  965 = 'S4_Warnings Default 965' | German: 'S4_Warnings German 965' | French: 'S4_Warnings French 965'
  966 = 'S4_Warnings Default 966' | German: 'S4_Warnings German 966' | French: 'S4_Warnings French 966'
  967 = 'S4_Warnings Default 967' | German: 'S4_Warnings German 967' | French: 'S4_Warnings French 967'
  968 = 'S4_Warnings Default 968' | German: 'S4_Warnings German 968' | French: 'S4_Warnings French 968'
  969 = 'S4_Warnings Default 969' | German: 'S4_Warnings German 969' | French: 'S4_Warnings French 969'
  970 = 'S4_Warnings Default 970' | German: 'S4_Warnings German 970' | French: 'S4_Warnings French 970'
  971 = 'S4_Warnings Default 971' | German: 'S4_Warnings German 971' | French: 'S4_Warnings French 971'
  972 = 'S4_Warnings Default 972' | German: 'S4_Warnings German 972' | French: 'S4_Warnings French 972'
  973 = 'S4_Warnings Default 973' | German: 'S4_Warnings German 973' | French: 'S4_Warnings French 973'
  974 = 'S4_Warnings Default 974' | German: 'S4_Warnings German 974' | French: 'S4_Warnings French 974'
  975 = 'S4_Warnings Default 975' | German: 'S4_Warnings German 975' | French: 'S4_Warnings French 975'
  976 = 'S4_Warnings Default 976' | German: 'S4_Warnings German 976' | French: 'S4_Warnings French 976'
  977 = 'S4_Warnings Default 977' | German: 'S4_Warnings German 977' | French: 'S4_Warnings French 977'
  978 = 'S4_Warnings Default 978' | German: 'S4_Warnings German 978' | French: 'S4_Warnings French 978'
  979 = 'S4_Warnings Default 979' | German: 'S4_Warnings German 979' | French: 'S4_Warnings French 979'
  980 = 'S4_Warnings Default 980' | German: 'S4_Warnings German 980' | French: 'S4_Warnings French 980'
  981 = 'S4_Warnings Default 981' | German: 'S4_Warnings German 981' | French: 'S4_Warnings French 981'
  982 = 'S4_Warnings Default 982' | German: 'S4_Warnings German 982' | French: 'S4_Warnings French 982'
  983 = 'S4_Warnings Default 983' | German: 'S4_Warnings German 983' | French: 'S4_Warnings French 983'
  984 = 'S4_Warnings Default 984' | German: 'S4_Warnings German 984' | French: 'S4_Warnings French 984'
  985 = 'S4_Warnings Default 985' | German: 'S4_Warnings German 985' | French: 'S4_Warnings French 985'
  986 = 'S4_Warnings Default 986' | German: 'S4_Warnings German 986' | French: 'S4_Warnings French 986'
  987 = 'S4_Warnings Default 987' | German: 'S4_Warnings German 987' | French: 'S4_Warnings French 987'
  988 = 'S4_Warnings Default 988' | German: 'S4_Warnings German 988' | French: 'S4_Warnings French 988'
  989 = 'S4_Warnings Default 989' | German: 'S4_Warnings German 989' | French: 'S4_Warnings French 989'
  990 = 'S4_Warnings Default 990' | German: 'S4_Warnings German 990' | French: 'S4_Warnings French 990'
  991 = 'S4_Warnings Default 991' | German: 'S4_Warnings German 991' | French: 'S4_Warnings French 991'
  992 = 'S4_Warnings Default 992' | German: 'S4_Warnings German 992' | French: 'S4_Warnings French 992'
  993 = 'S4_Warnings Default 993' | German: 'S4_Warnings German 993' | French: 'S4_Warnings French 993'
  994 = 'S4_Warnings Default 994' | German: 'S4_Warnings German 994' | French: 'S4_Warnings French 994'
  995 = 'S4_Warnings Default 995' | German: 'S4_Warnings German 995' | French: 'S4_Warnings French 995'
  996 = 'S4_Warnings Default 996' | German: 'S4_Warnings German 996' | French: 'S4_Warnings French 996'
  997 = 'S4_Warnings Default 997' | German: 'S4_Warnings German 997' | French: 'S4_Warnings French 997'
  998 = 'S4_Warnings Default 998' | German: 'S4_Warnings German 998' | French: 'S4_Warnings French 998'
  999 = 'S4_Warnings Default 999' | German: 'S4_Warnings German 999' | French: 'S4_Warnings French 999'
  1000 = 'S4_Warnings Default 1000' | German: 'S4_Warnings German 1000' | French: 'S4_Warnings French 1000'
   = ''
END_TEXTLIST

(* stored: Version 1.1.0.1, ProductVersion 3.1.4024.12
   TextList S4_Warnings: Id {b50b5de8-5ee3-4d5f-8803-3559b9c62b9a} *)
